// TIA Portal V15.1 export
// export: Created 2026-01-09T13:45:11.7607581Z, ExportSetting WithDefaults, WithReadOnly, DisplayName Totally Integrated Automation Portal, DisplayVersion V15.1 Update 8, DisplayName TIA Portal Openness, DisplayVersion V15.1 Update 8, DisplayName STEP 7 Professional, DisplayVersion V15.1 Update 8, DisplayName WinCC Advanced, DisplayVersion V15.1 Update 8
DATA_BLOCK "C#6_WD_CALIB"   // DB6
{ S7_Optimized_Access := 'FALSE' }
VERSION : 0.1
// stored: AutoNumber true, CodeModifiedDate 2026-01-01T14:21:06.6662125Z, CompileDate 2026-01-04T03:21:25.721467Z, CreationDate 2024-10-12T12:36:08.0193576Z, DBAccessibleFromOPCUA true, InterfaceModifiedDate 2026-01-01T14:21:06.6662125Z, IsConsistent true, IsKnowHowProtected false, IsOnlyStoredInLoadMemory false, IsPLCDB false, IsWriteProtectedInAS false, ModifiedDate 2026-01-01T14:21:06.6662125Z, ParameterModified 2026-01-01T14:21:06.6662125Z, StructureModified 2026-01-01T14:21:06.6662125Z
   VAR RETAIN
      KL_ZERO_AG1 : Real;   // Khối lượng chỉnh 0 cân AG1
      KL_SPAN_AG1 : Real;   // Khối lượng chỉnh tải cân AG1
      KL_ZERO_FD1 : Real;   // Khối lượng chỉnh 0 cân FD1
      KL_SPAN_FD1 : Real;   // Khối lượng chỉnh tải cân FD1
      KL_ZERO_AP1 : Real;   // Khối lượng chỉnh 0 cân AP1
      KL_SPAN_AP1 : Real;   // Khối lượng chỉnh tải cân AP1
      KL_ZERO_SB1 : Real;   // Khối lượng chỉnh 0 cân SB1
      KL_SPAN_SB1 : Real;   // Khối lượng chỉnh tải cân SB1
      ZERO_TEMP_TS : Real;   // Nhiệt độ T1 tan sấy
      SPAN_TEMP_TS : Real;   // Nhiệt độ T2 tan sấy
      ZERO_TEMP_AG : Real;   // Nhiệt độ T1 Cốt liệu Agg
      SPAN_TEMP_AG : Real;   // Nhiệt độ T2 Cốt kiệu Agg
      ZERO_TEMP_AP : Real;   // Nhiệt độ T1 Nhựa
      SPAN_TEMP_AP : Real;   // Nhiệt độ T2 Nhựa
      ZERO_TEMP_TL : Real;   // Nhiệt độ T1 Túi lọc
      SPAN_TEMP_TL : Real;   // Nhiệt độ T2 Túi lọc
      HS_AG1 : Real;   // Hệ số cân Ag1
      HS_FD1 : Real;   // Hệ số cân FD1
      HS_AP1 : Real;   // Hệ số cân AP1
      HS_SB1 : Real;   // Hệ số cân SB1
      "HS_TEMP TS" : Real;   // Hệ số nhiệt độ 1
      "HS_TEMP AG" : Real;   // Hệ số nhiệt độ 2
      "HS_TEMP AP" : Real;   // Hệ số nhiệt độ 3
      "HS_TEMP TL" : Real;   // Hệ số nhiệt độ 4
      XUNG_AG1 : Real;   // Đọc xung AG1
      XUNG_FD1 : Real;   // Đọc xung FD1
      XUNG_AP1 : Real;   // Đọc xung AP1
      XUNG_SB1 : Real;   // Đọc xung SB1
      XUNG_TEMP_TS : Real;   // Đọc xung nhiệt độ tan sấy
      XUNG_TEMP_AG : Real;   // Đọc xung nhiệt độ AGG
      XUNG_TEMP_AP : Real;   // Đọc xung nhiệt độ nhựa
      XUNG_TEMP_TL : Real;   // Đọc xung nhiệt độ túi lọc
      KLT_AG1 : Real;   // Đọc khối lượng cân AG
      KLT_FD1 : Real;   // Đọc khối lượng cân FD
      KLT_AP1 : Real;   // Đọc khối lượng cân AP
      KLT_SB1 : Real;   // Đọc khối lượng cân SBS
      NDT_TS : Real;   // Đọc nhiệt độ tan sấy
      NDT_AG : Real;   // Đọc nhiệt độ cốt liệu
      NDT_AP : Real;   // Đọc nhiệt độ nhựa
      NDT_TL : Real;   // Đọc nhiệt độ túi lọc bụi
      HMI_Manual_Pulse : Bool;
      KL_ZERO_IND_AGG1 : Real;
      KL_SPAN_IND_AGG1 : Real;
      HS_IND_AGG1 : Real;
      XUNG_IND_AGG1 : Real;
      KLT_IND_AGG1 : Real;
      KL_ZERO_IND_AGG2 : Real;
      KL_SPAN_IND_AGG2 : Real;
      HS_IND_AGG2 : Real;
      XUNG_IND_AGG2 : Real;
      KLT_IND_AGG2 : Real;
      KL_ZERO_IND_AGG3 : Real;
      KL_SPAN_IND_AGG3 : Real;
      HS_IND_AGG3 : Real;
      XUNG_IND_AGG3 : Real;
      KLT_IND_AGG3 : Real;
      KL_ZERO_IND_AGG4 : Real;
      KL_SPAN_IND_AGG4 : Real;
      HS_IND_AGG4 : Real;
      XUNG_IND_AGG4 : Real;
      KLT_IND_AGG4 : Real;
      KL_ZERO_IND_AGG5 : Real;
      KL_SPAN_IND_AGG5 : Real;
      HS_IND_AGG5 : Real;
      XUNG_IND_AGG5 : Real;
      KLT_IND_AGG5 : Real;
   END_VAR
BEGIN
END_DATA_BLOCK
